RoboDK station: RoboticsABB.rdk

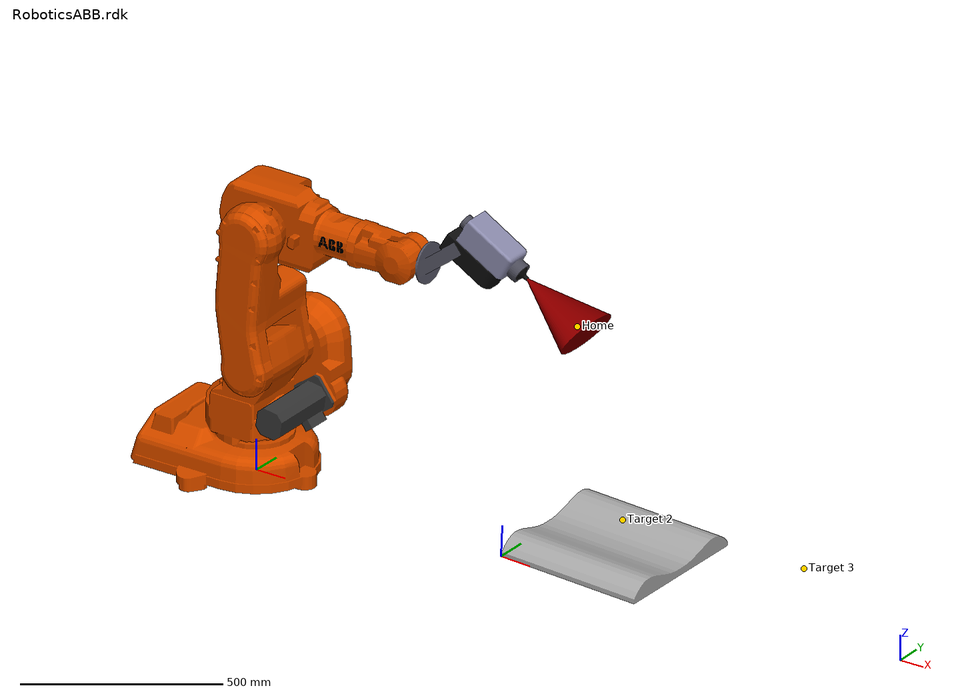
[picture v0: the station drawn from its stored meshes, robots at their saved joint values, targets as dots, program paths as lines]
Station RoboticsABB (saved by RoboDK 5.7.1). Poses are relative to the parent item; angles as X-Y-Z fixed-axis rotations.
  - frame ABB IRB 140-6/0.8 Base at (-682.05, 0, 0) mm
    - robot ABB IRB 140-6/0.8: 6 axes, payload 6 kg, reach 810 mm, repeatability 0.03 mm, weight 98 kg
        modified DH rows (alpha deg, a mm, theta deg, d mm): 0, 0, 0, 352; -90, 70, -90, 0; 0, 360, 0, 0; -90, 0, 0, 380; 90, 0, 0, 0; -90, 0, 180, 65
        joint limits [-180, -90, -230, -200, -120, -400] to [180, 110, 50, 200, 120, 400]; home [0, 0, 0, 0, 0, 0]; saved at [0, 0, 0, 0, 0, 0]
      - tool Paint gun, TCP at (50, 0, 450) mm, rotated rx 0 ry 30 rz 0 deg, size 203.2 x 279.7 x 471.5 mm
    - target Home (Cartesian target) at (965, 0, 662) mm, rotated rx -180 ry 60 rz -180 deg; joints [0, 0, 0, 0, 0, 0] of ABB IRB 140-6/0.8
  - frame Frame 2 at (0, 77.85, -77.58) mm, rotated rx 0 ry 2.63 rz 0 deg
    - object Object Inspection at (0, 0, 0) mm, size 400 x 400 x 46.2 mm, geometry from Object Inspection.stp
    - target Target 2 (Cartesian target) at (218.01, 205.02, 90.75) mm, rotated rx -177.58 ry 3.27 rz 168.82 deg; joints [26.735, 65.349, -60.62, -22.899, 63.57, 43.47] of ABB IRB 140-6/0.8
    - target Target 3 (Cartesian target) at (743.22, 233.25, 116.52) mm, rotated rx 171.03 ry 11.08 rz 138.39 deg; joints [38.73, 29.5, -8.95, -45.57, 60.76, 102.03] of ABB IRB 140-6/0.8
